{attribute 'qualified_only'}
{attribute 'strict'}
{attribute 'tostring'}
TYPE eCOAlarmStatus :
(
	Error			:= 0,
	Normal 			:= 1,
	WarningLevel1 	:= 2,
	WarningLevel2 	:= 3,
	Alarm 			:= 4
);
END_TYPE

(* stored: Version 1.1.0.1, ProductVersion 3.1.4026.18
   DUT eCOAlarmStatus: Id {406822b2-650f-4fa9-aaa4-84cc6bc1ef5f} *)
